FUNCTION_BLOCK FB_ADD
VAR_INPUT
	in1,in2;INT;
END_VAR
VAR_OUTPUT
	out:INT;
END_VAR
VAR
END_VAR

out:=in1+in2;

END_FUNCTION_BLOCK

(* stored: Version 1.1.0.1, ProductVersion 3.1.4024.3
   POU FB_ADD: Id {6814feed-ecc9-4f5d-82ff-a8d42cb9b61e}, SpecialFunc None *)
